INTERFACE I_EventTarget EXTENDS __SYSTEM.IQueryInterface

METHOD PUBLIC Emit
VAR_INPUT
	EventName : T_MaxString;
	Event : I_Event;
END_VAR
END_METHOD

END_INTERFACE

(* stored: Version 1.1.0.1, ProductVersion 3.1.4024.12
   Itf I_EventTarget: Id {2428aaaf-eea6-4643-bd6f-1b4bb59ac2e9}
   Method Emit: Id {2a89147a-333d-4199-bc9e-1f5968cfe90f} *)
